KUKA KRL program: ho_st600_r1_bolha.src, ho_st600_r1_bolha.dat

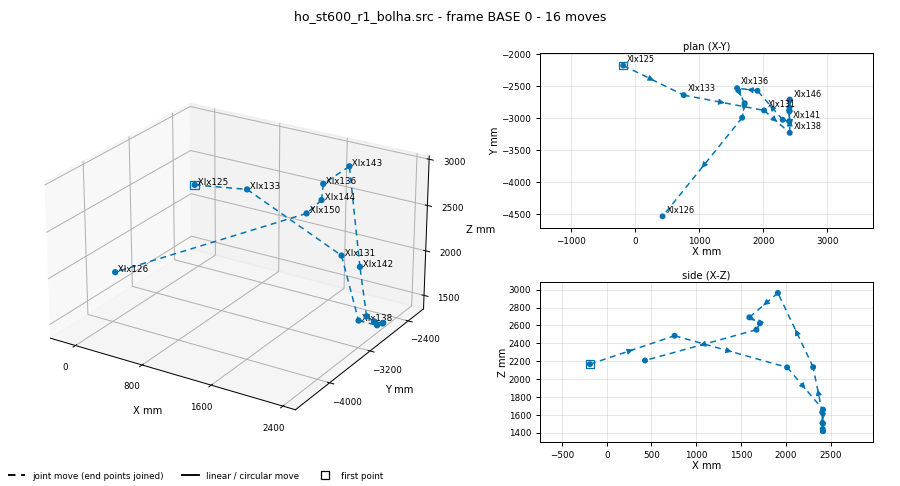
[picture p0: tool path of ho_st600_r1_bolha.src in frame BASE 0, 16 of 16 moves have a stored position in this frame; points joined in program order, loops and branches not executed]
--- ho_st600_r1_bolha.src ---
&ACCESS RVO1
&REL 2
&COMMENT Pega traseira ACCELO BOLHA
&PARAM DISKPATH = KRC:\R1\Program
DEF ho_st600_r1_Bolha( )
;FOLD INI
  ;FOLD BASISTECH INI
    GLOBAL INTERRUPT DECL 3 WHEN $STOPMESS==TRUE DO IR_STOPM ( )
    INTERRUPT ON 3
    BAS (#INITMOV,0 )
  ;ENDFOLD (BASISTECH INI)
;FOLD GRIPPERTECH INI
USER_GRP(0,DUMMY,DUMMY,GDEFAULT)
;ENDFOLD (GRIPPERTECH INI)
  ;FOLD USER INI
    ;Make your modifications here

  ;ENDFOLD (USER INI)
;ENDFOLD (INI)

; Caracterização dos meios de produção:
; Changes: Pega Traseira Accelo
; Versão Atual: 21/07/2015
; Name: P13.050-R1

chk_w7_wechs_ok ( )  ;CHECK GRIPPER TRASEIRO ACCELO


;FOLD PTP lx125 Vel=100 % PDAT8 Tool[7]:Painel Traseiro Accelo Base[0];%{PE}%R 8.2.20,%MKUKATPBASIS,%CMOVE,%VPTP,%P 1:PTP, 2:lx125, 3:, 5:100, 7:PDAT8
$BWDSTART=FALSE
PDAT_ACT=PPDAT8
FDAT_ACT=Flx125
BAS(#PTP_PARAMS,100)
PTP Xlx125
;ENDFOLD


;** SETUP DOS GRAMPOS PARA A BOLHA

;FOLD OUT 251 'Y2VR_FECHA_Accelo_Bolha' State=TRUE ;%{PE}%R 8.2.20,%MKUKATPBASIS,%COUT,%VOUTX,%P 2:251, 3:Y2VR_FECHA_Accelo_Bolha, 5:TRUE, 6:
$OUT[251]=TRUE
;ENDFOLD
;FOLD WAIT FOR ( IN 250 'Z2.1 - Grampo Avancado - Accelo Bolha' ) AND ( IN 252 'Z2.2 - Grampo Avancado - Accelo Bolha' );%{PE}%R 8.2.20,%MKUKATPBASIS,%CEXT_WAIT_FOR,%VEXT_WAIT_FOR,%P 2:, 4:, 5:$IN, 6:250, 7:Z2.1 - Grampo Avancado - Accelo Bolha, 9:AND, 10:, 12:, 13:$IN, 14:252, 15:Z2.2 - Grampo Avancado - Accelo Bolha, 17:
WAIT FOR  ( $IN[250] ) AND ( $IN[252] )
;ENDFOLD
;FOLD OUT 249 'Y1VR_FECHA_Accelo' State=TRUE ;%{PE}%R 8.2.20,%MKUKATPBASIS,%COUT,%VOUTX,%P 2:249, 3:Y1VR_FECHA_Accelo, 5:TRUE, 6:
$OUT[249]=TRUE
;ENDFOLD
;FOLD WAIT FOR ( IN 246 'Z1.2 - Grampo Avancado - Accelo - Traseiro' ) AND ( IN 248 'Z1.1 - Grampo Avancado - Accelo - Traseiro' );%{PE}%R 8.2.20,%MKUKATPBASIS,%CEXT_WAIT_FOR,%VEXT_WAIT_FOR,%P 2:, 4:, 5:$IN, 6:246, 7:Z1.2 - Grampo Avancado - Accelo - Traseiro, 9:AND, 10:, 12:, 13:$IN, 14:248, 15:Z1.1 - Grampo Avancado - Accelo - Traseiro, 17:
WAIT FOR  ( $IN[246] ) AND ( $IN[248] )
;ENDFOLD
;FOLD OUT 254 'Y3VR_RECUA_CILINDRO_Accelo/Bolha' State=TRUE ;%{PE}%R 8.2.20,%MKUKATPBASIS,%COUT,%VOUTX,%P 2:254, 3:Y3VR_RECUA_CILINDRO_Accelo/Bolha, 5:TRUE, 6:
$OUT[254]=TRUE
;ENDFOLD


;FOLD PTP lx133 Vel=100 % PDAT0 Tool[7]:Painel Traseiro Accelo Base[0];%{PE}%R 8.2.20,%MKUKATPBASIS,%CMOVE,%VPTP,%P 1:PTP, 2:lx133, 3:, 5:100, 7:PDAT0
$BWDSTART=FALSE
PDAT_ACT=PPDAT0
FDAT_ACT=Flx133
BAS(#PTP_PARAMS,100)
PTP Xlx133
;ENDFOLD

;FOLD WAIT FOR ( IN 253 'Z3.1 - Cilindro Recuado - Accelo' ) AND ( IN 255 'Z3.2 - Cilindro Recuado - Accelo' );%{PE}%R 8.2.20,%MKUKATPBASIS,%CEXT_WAIT_FOR,%VEXT_WAIT_FOR,%P 2:, 4:, 5:$IN, 6:253, 7:Z3.1 - Cilindro Recuado - Accelo, 9:AND, 10:, 12:, 13:$IN, 14:255, 15:Z3.2 - Cilindro Recuado - Accelo, 17:
WAIT FOR  ( $IN[253] ) AND ( $IN[255] )
;ENDFOLD
;FOLD OUT 251 'Y2VR_FECHA_Accelo_Bolha' State=FALSE ;%{PE}%R 8.2.20,%MKUKATPBASIS,%COUT,%VOUTX,%P 2:251, 3:Y2VR_FECHA_Accelo_Bolha, 5:FALSE, 6:
$OUT[251]=FALSE
;ENDFOLD
;FOLD WAIT Time=0.5 sec;%{PE}%R 8.2.20,%MKUKATPBASIS,%CWAIT,%VWAIT,%P 3:0.5
WAIT SEC 0.5
;ENDFOLD
;FOLD OUT 252 'Y2VR_ABRE_Accelo_Bolha' State=TRUE ;%{PE}%R 8.2.20,%MKUKATPBASIS,%COUT,%VOUTX,%P 2:252, 3:Y2VR_ABRE_Accelo_Bolha, 5:TRUE, 6:
$OUT[252]=TRUE
;ENDFOLD
;FOLD WAIT FOR ( IN 249 'Z2.1 - Grampo Recuado - Accelo Bolha' ) AND ( IN 251 'Z2.2 - Grampo Recuado - Accelo Bolha' );%{PE}%R 8.2.20,%MKUKATPBASIS,%CEXT_WAIT_FOR,%VEXT_WAIT_FOR,%P 2:, 4:, 5:$IN, 6:249, 7:Z2.1 - Grampo Recuado - Accelo Bolha, 9:AND, 10:, 12:, 13:$IN, 14:251, 15:Z2.2 - Grampo Recuado - Accelo Bolha, 17:
WAIT FOR  ( $IN[249] ) AND ( $IN[251] )
;ENDFOLD



;FOLD PTP lx131 CONT Vel=75 % PDAT14 Tool[7]:Painel Traseiro Accelo Base[0];%{PE}%R 8.2.20,%MKUKATPBASIS,%CMOVE,%VPTP,%P 1:PTP, 2:lx131, 3:C_DIS, 5:75, 7:PDAT14
$BWDSTART=FALSE
PDAT_ACT=PPDAT14
FDAT_ACT=Flx131
BAS(#PTP_PARAMS,75)
PTP Xlx131 C_DIS
;ENDFOLD

;FOLD PTP lx138 Vel=75 % PDAT21 Tool[7]:Painel Traseiro Accelo Base[0];%{PE}%R 8.2.20,%MKUKATPBASIS,%CMOVE,%VPTP,%P 1:PTP, 2:lx138, 3:, 5:75, 7:PDAT21
$BWDSTART=FALSE
PDAT_ACT=PPDAT21
FDAT_ACT=Flx138
BAS(#PTP_PARAMS,75)
PTP Xlx138
;ENDFOLD

;FOLD OUT 3352 'R1 busca traseira' State=TRUE ;%{PE}%R 8.2.20,%MKUKATPBASIS,%COUT,%VOUTX,%P 2:3352, 3:R1 busca traseira, 5:TRUE, 6:
$OUT[3352]=TRUE
;ENDFOLD
;FOLD WAIT FOR ( IN 3352 'Aguarda lib. Buscar traseira' );%{PE}%R 8.2.20,%MKUKATPBASIS,%CEXT_WAIT_FOR,%VEXT_WAIT_FOR,%P 2:, 4:, 5:$IN, 6:3352, 7:Aguarda lib. Buscar traseira, 9:
WAIT FOR  ( $IN[3352] )
;ENDFOLD
;FOLD OUT 3352 'R1 busca traseira' State=FALSE ;%{PE}%R 8.2.20,%MKUKATPBASIS,%COUT,%VOUTX,%P 2:3352, 3:R1 busca traseira, 5:FALSE, 6:
$OUT[3352]=FALSE
;ENDFOLD

;FOLD PTP lx124 CONT Vel=100 % PDAT7 Tool[7]:Painel Traseiro Accelo Base[0];%{PE}%R 8.2.20,%MKUKATPBASIS,%CMOVE,%VPTP,%P 1:PTP, 2:lx124, 3:C_DIS, 5:100, 7:PDAT7
$BWDSTART=FALSE
PDAT_ACT=PPDAT7
FDAT_ACT=Flx124
BAS(#PTP_PARAMS,100)
PTP Xlx124 C_DIS
;ENDFOLD
;FOLD PTP lx146 CONT Vel=100 % P_OLP5 Tool[7]:Painel Traseiro Accelo Base[0];%{PE}%R 8.2.20,%MKUKATPBASIS,%CMOVE,%VPTP,%P 1:PTP, 2:lx146, 3:C_DIS, 5:100, 7:P_OLP5
$BWDSTART=FALSE
PDAT_ACT=PP_OLP5
FDAT_ACT=Flx146
BAS(#PTP_PARAMS,100)
PTP Xlx146 C_DIS
;ENDFOLD

;FOLD OUT 3342 'Fora area externa' State=FALSE ;%{PE}%R 8.2.20,%MKUKATPBASIS,%COUT,%VOUTX,%P 2:3342, 3:Fora area externa, 5:FALSE, 6:
$OUT[3342]=FALSE
;ENDFOLD

;FOLD ; PONTO DE PEGA DA TRASEIRA ACCELO;%{PE}%R 8.2.20,%MKUKATPBASIS,%CCOMMENT,%VNORMAL,%P 2:PONTO  DE  PEGA  DA  TRASEIRA  ACCELO
;ENDFOLD
;FOLD LIN Xlx145  Vel=0.25 m/s L_OLP1 Tool[7]" " Base[0] ;%{PE}%R8.2,%MKUKATPBASIS,%CMOVE,%VLIN,%P 1:LIN, 2:lx145, 3:, 5:0.25, 7:L_OLP1
$BWDSTART = FALSE
LDAT_ACT= LL_OLP1
FDAT_ACT= Flx145
BAS(#CP_PARAMS,0.25)
LIN Xlx145
;ENDFOLD

IF (NOT(GHOST())) THEN
;FOLD WAIT FOR ( IN 241 'Presenca de peca 1 Accelo Bolha TRASEIRO' ) AND ( IN 242 'Presenca de peca 2 Accelo Bolha TRASEIRO' );%{PE}%R 8.2.20,%MKUKATPBASIS,%CEXT_WAIT_FOR,%VEXT_WAIT_FOR,%P 2:, 4:, 5:$IN, 6:241, 7:Presenca de peca 1 Accelo Bolha TRASEIRO, 9:AND, 10:, 12:, 13:$IN, 14:242, 15:Presenca de peca 2 Accelo Bolha TRASEIRO, 17:
WAIT FOR  ( $IN[241] ) AND ( $IN[242] )
;ENDFOLD
ENDIF


;FOLD OUT 252 'Y2VR_ABRE_Accelo_Bolha' State=FALSE ;%{PE}%R 8.2.20,%MKUKATPBASIS,%COUT,%VOUTX,%P 2:252, 3:Y2VR_ABRE_Accelo_Bolha, 5:FALSE, 6:
$OUT[252]=FALSE
;ENDFOLD

;FOLD OUT 251 'Y2VR_FECHA_Accelo_Bolha' State=TRUE ;%{PE}%R 8.2.20,%MKUKATPBASIS,%COUT,%VOUTX,%P 2:251, 3:Y2VR_FECHA_Accelo_Bolha, 5:TRUE, 6:
$OUT[251]=TRUE
;ENDFOLD
;FOLD WAIT FOR ( IN 250 'Z2.1 - Grampo Avancado - Accelo Bolha' ) AND ( IN 252 'Z2.2 - Grampo Avancado - Accelo Bolha' );%{PE}%R 8.2.20,%MKUKATPBASIS,%CEXT_WAIT_FOR,%VEXT_WAIT_FOR,%P 2:, 4:, 5:$IN, 6:250, 7:Z2.1 - Grampo Avancado - Accelo Bolha, 9:AND, 10:, 12:, 13:$IN, 14:252, 15:Z2.2 - Grampo Avancado - Accelo Bolha, 17:
WAIT FOR  ( $IN[250] ) AND ( $IN[252] )
;ENDFOLD

;FOLD OUT 248 'Liga_Sugador_Accelo_Bolha' State=TRUE ;%{PE}%R 8.2.20,%MKUKATPBASIS,%COUT,%VOUTX,%P 2:248, 3:Liga_Sugador_Accelo_Bolha, 5:TRUE, 6:
$OUT[248]=TRUE
;ENDFOLD
;FOLD WAIT FOR ( IN 259 'Vacuo1_Accelo_Bolha' ) AND ( IN 260 'Vacuo2_Accelo_Bolha' );%{PE}%R 8.2.20,%MKUKATPBASIS,%CEXT_WAIT_FOR,%VEXT_WAIT_FOR,%P 2:, 4:, 5:$IN, 6:259, 7:Vacuo1_Accelo_Bolha, 9:AND, 10:, 12:, 13:$IN, 14:260, 15:Vacuo2_Accelo_Bolha, 17:
WAIT FOR  ( $IN[259] ) AND ( $IN[260] )
;ENDFOLD

;FOLD OUT 257 'Liga_Magnetico_Accelo_Bolha' State=TRUE ;%{PE}%R 8.2.20,%MKUKATPBASIS,%COUT,%VOUTX,%P 2:257, 3:Liga_Magnetico_Accelo_Bolha, 5:TRUE, 6:
$OUT[257]=TRUE
;ENDFOLD




IF (NOT(GHOST())) THEN
ENDIF


;FOLD OUT 3349 'R1 pegou peça' State=TRUE ;%{PE}%R 8.2.20,%MKUKATPBASIS,%COUT,%VOUTX,%P 2:3349, 3:R1 pegou peça, 5:TRUE, 6:
$OUT[3349]=TRUE
;ENDFOLD
;FOLD OUT 3350 'Solicita lib sair magazine' State=TRUE ;%{PE}%R 8.2.20,%MKUKATPBASIS,%COUT,%VOUTX,%P 2:3350, 3:Solicita lib sair magazine, 5:TRUE, 6:
$OUT[3350]=TRUE
;ENDFOLD
;FOLD WAIT FOR ( IN 3349 'Aguarda lib sair magazine' );%{PE}%R 8.2.20,%MKUKATPBASIS,%CEXT_WAIT_FOR,%VEXT_WAIT_FOR,%P 2:, 4:, 5:$IN, 6:3349, 7:Aguarda lib sair magazine, 9:
WAIT FOR  ( $IN[3349] )
;ENDFOLD
;FOLD OUT 3350 'Solicita lib sair magazine' State=FALSE ;%{PE}%R 8.2.20,%MKUKATPBASIS,%COUT,%VOUTX,%P 2:3350, 3:Solicita lib sair magazine, 5:FALSE, 6:
$OUT[3350]=FALSE
;ENDFOLD

;FOLD LIN Xlx149  Vel=0.25 m/s L_OLP2 Tool[7]" " Base[0] ;%{PE}%R8.2,%MKUKATPBASIS,%CMOVE,%VLIN,%P 1:LIN, 2:lx149, 3:, 5:0.25, 7:L_OLP2
$BWDSTART = FALSE
LDAT_ACT= LL_OLP2
FDAT_ACT= Flx149
BAS(#CP_PARAMS,0.25)
LIN Xlx149
;ENDFOLD

;FOLD PTP lx134 CONT Vel=100 % PDAT17 Tool[7]:Painel Traseiro Accelo Base[0];%{PE}%R 8.2.20,%MKUKATPBASIS,%CMOVE,%VPTP,%P 1:PTP, 2:lx134, 3:C_DIS, 5:100, 7:PDAT17
$BWDSTART=FALSE
PDAT_ACT=PPDAT17
FDAT_ACT=Flx134
BAS(#PTP_PARAMS,100)
PTP Xlx134 C_DIS
;ENDFOLD


;FOLD PTP lx141 CONT Vel=100 % PDAT24 Tool[7]:Painel Traseiro Accelo Base[0];%{PE}%R 8.2.20,%MKUKATPBASIS,%CMOVE,%VPTP,%P 1:PTP, 2:lx141, 3:C_DIS, 5:100, 7:PDAT24
$BWDSTART=FALSE
PDAT_ACT=PPDAT24
FDAT_ACT=Flx141
BAS(#PTP_PARAMS,100)
PTP Xlx141 C_DIS
;ENDFOLD

;FOLD PTP lx142 CONT Vel=100 % PDAT25 Tool[7]:Painel Traseiro Accelo Base[0];%{PE}%R 8.2.20,%MKUKATPBASIS,%CMOVE,%VPTP,%P 1:PTP, 2:lx142, 3:C_DIS, 5:100, 7:PDAT25
$BWDSTART=FALSE
PDAT_ACT=PPDAT25
FDAT_ACT=Flx142
BAS(#PTP_PARAMS,100)
PTP Xlx142 C_DIS
;ENDFOLD


;FOLD PTP lx143 CONT Vel=100 % PDAT26 Tool[7]:Painel Traseiro Accelo Base[0];%{PE}%R 8.2.20,%MKUKATPBASIS,%CMOVE,%VPTP,%P 1:PTP, 2:lx143, 3:C_DIS, 5:100, 7:PDAT26
$BWDSTART=FALSE
PDAT_ACT=PPDAT26
FDAT_ACT=Flx143
BAS(#PTP_PARAMS,100)
PTP Xlx143 C_DIS
;ENDFOLD

;FOLD PTP lx136 CONT Vel=100 % PDAT19 Tool[7]:Painel Traseiro Accelo Base[0];%{PE}%R 8.2.20,%MKUKATPBASIS,%CMOVE,%VPTP,%P 1:PTP, 2:lx136, 3:C_DIS, 5:100, 7:PDAT19
$BWDSTART=FALSE
PDAT_ACT=PPDAT19
FDAT_ACT=Flx136
BAS(#PTP_PARAMS,100)
PTP Xlx136 C_DIS
;ENDFOLD

;FOLD PTP lx144 CONT Vel=100 % PDAT27 Tool[7]:Painel Traseiro Accelo Base[0];%{PE}%R 8.2.20,%MKUKATPBASIS,%CMOVE,%VPTP,%P 1:PTP, 2:lx144, 3:C_DIS, 5:100, 7:PDAT27
$BWDSTART=FALSE
PDAT_ACT=PPDAT27
FDAT_ACT=Flx144
BAS(#PTP_PARAMS,100)
PTP Xlx144 C_DIS
;ENDFOLD

;FOLD PTP lx150 CONT Vel=100 % P_OLP6 Tool[7]:Painel Traseiro Accelo Base[0];%{PE}%R8.2,%MKUKATPBASIS,%CMOVE,%VPTP,%P 1:PTP, 2:lx150, 3:C_DIS, 5:100, 7:P_OLP6
$BWDSTART = FALSE
PDAT_ACT= PP_OLP6
FDAT_ACT= Flx150
BAS(#PTP_PARAMS,100)
PTP Xlx150 C_DIS
;ENDFOLD
;FOLD PTP lx126 CONT Vel=100 % PDAT9 Tool[7]:Painel Traseiro Accelo Base[0];%{PE}%R 8.2.20,%MKUKATPBASIS,%CMOVE,%VPTP,%P 1:PTP, 2:lx126, 3:C_DIS, 5:100, 7:PDAT9
$BWDSTART=FALSE
PDAT_ACT=PPDAT9
FDAT_ACT=Flx126
BAS(#PTP_PARAMS,100)
PTP Xlx126 C_DIS
;ENDFOLD

;FOLD OUT 3349 'R1 Pegou peca' State=TRUE ;%{PE}%R 8.2.20,%MKUKATPBASIS,%COUT,%VOUTX,%P 2:3349, 3:R1 Pegou peca, 5:TRUE, 6:
$OUT[3349]=TRUE
;ENDFOLD
;FOLD OUT 3342 'Fora area externa' State=TRUE ;%{PE}%R 8.2.20,%MKUKATPBASIS,%COUT,%VOUTX,%P 2:3342, 3:Fora area externa, 5:TRUE, 6:
$OUT[3342]=TRUE
;ENDFOLD

END

--- ho_st600_r1_bolha.dat ---
&ACCESS RVO1
&REL 2
&COMMENT Pega traseira ACCELO BOLHA
&PARAM DISKPATH = KRC:\R1\Program
DEFDAT  ho_st600_r1_Bolha
;FOLD EXTERNAL DECLARATIONS;%{PE}%MKUKATPBASIS,%CEXT,%VCOMMON,%P
;FOLD GRIPPERTECH EXT
EXT  H50 (INT  :IN,INT  :IN,INT  :IN,GRP_TYP  :IN )
;ENDFOLD (GRIPPERTECH EXT)
;FOLD SPOTTECH EXT
EXT  USERSPOT (S_COMMAND  :IN,SPOT_TYPE  :IN )
;ENDFOLD (SPOTTECH EXT)
;FOLD BASISTECH EXT;%{PE}%MKUKATPBASIS,%CEXT,%VEXT,%P
EXT  BAS (BAS_COMMAND  :IN,REAL  :IN )
DECL INT SUCCESS
;ENDFOLD (BASISTECH EXT)
;FOLD USER EXT;%{E}%MKUKATPUSER,%CEXT,%VEXT,%P
;Make your modifications here

;ENDFOLD (USER EXT)
;ENDFOLD (EXTERNAL DECLARATIONS)

;# ============ START PATH : bh_p13050r1_ltc_02 =============
DECL FDAT Flx146={TOOL_NO 7,BASE_NO 0,IPO_FRAME #BASE,POINT2[] " ",TQ_STATE FALSE}
DECL PDAT PP_OLP5={VEL 100.0,ACC 100.0,APO_DIST 0.0,APO_MODE #CDIS}
DECL E6POS Xlx146={X 2414.24609,Y -2720.17798,Z 1419.953,A 89.8186417,B -64.6082993,C 179.921097,S 2,T 11,E1 -3712.55103,E2 0.0,E3 0.0,E4 0.0,E5 0.0,E6 0.0}
DECL FDAT Flx145={TOOL_NO 7,BASE_NO 0,IPO_FRAME #BASE,POINT2[] " ",TQ_STATE FALSE}
DECL E6POS Xlx145={X 2414.01489,Y -2707.33691,Z 1420.96399,A 89.5057068,B -64.9538422,C -179.770599,S 2,T 11,E1 -3712.55493,E2 0.0,E3 0.0,E4 0.0,E5 0.0,E6 0.0}
DECL LDAT LL_OLP1={VEL 0.25,ACC 100.0,APO_DIST 0.0,APO_FAC 0.0}
DECL FDAT Flx149={TOOL_NO 7,BASE_NO 0,IPO_FRAME #BASE,POINT2[] " "}
DECL E6POS Xlx149={X 2413.25488,Y -2887.86401,Z 1505.32397,A 89.5048828,B -64.9540634,C -179.769699,S 2,T 11,E1 -3712.55688,E2 0.0,E3 0.0,E4 0.0,E5 0.0,E6 0.0}
DECL LDAT LL_OLP2={VEL 0.25,ACC 100.0,APO_DIST 0.0,APO_FAC 0.0}
DECL FDAT Flx150={TOOL_NO 7,BASE_NO 0,IPO_FRAME #BASE,POINT2[] " "}
DECL PDAT PP_OLP6={VEL 100.0,ACC 100.0,APO_DIST 100.0,APO_MODE #CDIS}
DECL E6POS Xlx150={X 1671.224,Y -2991.78491,Z 2552.60889,A 44.4150009,B -75.0324783,C 129.688202,S 2,T 3,E1 -2192.70093,E2 0.0,E3 0.0,E4 0.0,E5 0.0,E6 0.0}
DECL BASIS_SUGG_T LAST_BASIS={POINT1[] "P0                      ",POINT2[] "P0                      ",CP_PARAMS[] "CPDAT0                  ",PTP_PARAMS[] "PDAT0                   ",CONT[] "                        ",CP_VEL[] "2.0                     ",PTP_VEL[] " 100                    ",SYNC_PARAMS[] "SYNCDAT                 ",SPL_NAME[] "S0                      "}
DECL GRP_SUGG_T LAST_GRP={NUMBER[] "5                       ",STATE[] "1                       ",PARAMS[] "GDAT3                   "}
DECL GRP_TYP GGDAT1={G_APO #NO,GRP_TIME 0.200000003,CTRL #OFF,DLY 0,DST 1}
DECL GRP_TYP GGDAT2={G_APO #NO,GRP_TIME 0.200000003,CTRL #OFF,DLY 0,DST 1}
DECL GRP_TYP GGDAT3={G_APO #NO,GRP_TIME 0.200000003,CTRL #OFF,DLY 0,DST 1}
DECL PDAT PPDAT7={VEL 100.0,ACC 100.0,APO_DIST 100.0,APO_MODE #CDIS}
DECL E6POS Xlx124={X 2410.65894,Y -2831.65405,Z 1444.37695,A 89.8383408,B -65.6056671,C -179.489899,S 2,T 11,E1 -3712.54712,E2 0.0,E3 0.0,E4 0.0,E5 0.0,E6 0.0}
DECL FDAT Flx124={TOOL_NO 7,BASE_NO 0,IPO_FRAME #BASE,POINT2[] " ",TQ_STATE FALSE}
DECL GRP_TYP GCONT={G_APO #YES,GRP_TIME 0.0,CTRL #OFF,DLY 0,DST 0}
DECL PDAT PPDAT8={VEL 100.0,ACC 100.0,APO_DIST 100.0,APO_MODE #CDIS}
DECL E6POS Xlx125={X -187.007996,Y -2175.83301,Z 2167.93994,A 48.8575897,B -57.0335617,C -142.841705,S 2,T 3,E1 -3715.35498,E2 0.0,E3 0.0,E4 0.0,E5 0.0,E6 0.0}
DECL FDAT Flx125={TOOL_NO 7,BASE_NO 0,IPO_FRAME #BASE,POINT2[] " ",TQ_STATE FALSE}
DECL E6POS XLX126={X 427.047913,Y -4533.16797,Z 2209.23389,A -73.5128708,B -78.8541565,C -161.542206,S 6,T 18,E1 -2536.18188,E2 0.0,E3 0.0,E4 0.0,E5 0.0,E6 0.0}
DECL FDAT Flx126={TOOL_NO 7,BASE_NO 0,IPO_FRAME #BASE,POINT2[] " ",TQ_STATE FALSE}
DECL PDAT PPDAT9={VEL 100.0,ACC 100.0,APO_DIST 100.0,APO_MODE #CDIS}
DECL GRP_TYP GGDAT4={G_APO #NO,GRP_TIME 0.200000003,CTRL #OFF,DLY 0,DST 1}
DECL PDAT PPDAT14={VEL 100.0,ACC 100.0,APO_DIST 100.0,APO_MODE #CDIS}
DECL E6POS Xlx131={X 2013.56104,Y -2877.54102,Z 2132.77197,A 86.6203995,B -62.3385391,C -177.631393,S 2,T 11,E1 -3712.88208,E2 0.0,E3 0.0,E4 0.0,E5 0.0,E6 0.0}
DECL FDAT Flx131={TOOL_NO 7,BASE_NO 0,IPO_FRAME #BASE,POINT2[] " ",TQ_STATE FALSE}
DECL PDAT PPDAT15={VEL 100.0,ACC 100.0,APO_DIST 100.0,APO_MODE #CDIS}
DECL E6POS Xlx132={X 757.784119,Y -2638.58398,Z 2485.66089,A 86.4221573,B -61.0999107,C -174.462006,S 2,T 11,E1 -3713.53003,E2 0.0,E3 0.0,E4 0.0,E5 0.0,E6 0.0}
DECL FDAT Flx132={TOOL_NO 7,BASE_NO 0,IPO_FRAME #BASE,POINT2[] " ",TQ_STATE FALSE}
DECL E6POS XLX134={X 2408.49707,Y -2891.43506,Z 1510.60596,A 89.8388672,B -65.7432404,C -179.910995,S 2,T 11,E1 -3712.552,E2 0.0,E3 0.0,E4 0.0,E5 0.0,E6 0.0}
DECL FDAT Flx134={TOOL_NO 7,BASE_NO 0,IPO_FRAME #BASE,POINT2[] " ",TQ_STATE FALSE}
DECL PDAT PPDAT17={VEL 100.0,ACC 100.0,APO_DIST 100.0,APO_MODE #CDIS}
DECL E6POS XLX135={X 2079.61499,Y -2528.86206,Z 2745.854,A 122.505203,B -59.1623993,C 117.408401,S 2,T 11,E1 -3182.0481,E2 0.0,E3 0.0,E4 0.0,E5 0.0,E6 0.0}
DECL FDAT Flx135={TOOL_NO 7,BASE_NO 0,IPO_FRAME #BASE,POINT2[] " ",TQ_STATE FALSE}
DECL PDAT PPDAT18={VEL 100.0,ACC 80.0,APO_DIST 80.0,APO_MODE #CDIS}
DECL E6POS XLX136={X 1592.48901,Y -2529.09399,Z 2691.021,A 97.9955597,B -64.183548,C 126.372902,S 2,T 11,E1 -2840.72803,E2 0.0,E3 0.0,E4 0.0,E5 0.0,E6 0.0}
DECL FDAT Flx136={TOOL_NO 7,BASE_NO 0,IPO_FRAME #BASE,POINT2[] " ",TQ_STATE FALSE}
DECL PDAT PPDAT19={VEL 100.0,ACC 80.0,APO_DIST 80.0,APO_MODE #CDIS}
DECL GRP_TYP GGDAT5={G_APO #NO,GRP_TIME 0.200000003,CTRL #OFF,DLY 0,DST 1}
DECL GRP_TYP GGDAT6={G_APO #NO,GRP_TIME 0.200000003,CTRL #OFF,DLY 0,DST 1}
DECL E6POS XLX138={X 2415.00293,Y -3227.64795,Z 1660.75,A 90.586319,B -65.2316589,C 179.779297,S 2,T 11,E1 -3712.55103,E2 0.0,E3 0.0,E4 0.0,E5 0.0,E6 0.0}
DECL FDAT Flx138={TOOL_NO 7,BASE_NO 0,IPO_FRAME #BASE,POINT2[] " ",TQ_STATE FALSE}
DECL PDAT PPDAT21={VEL 100.0,ACC 100.0,APO_DIST 100.0,APO_MODE #CDIS}
DECL E6POS XLX139={X 4758.36914,Y -8491.97852,Z -555.414185,A -47.7297401,B -59.6328011,C 156.117004,S 2,T 3,E1 -1239.23804,E2 0.0,E3 0.0,E4 0.0,E5 0.0,E6 0.0}
DECL FDAT Flx139={TOOL_NO 7,BASE_NO 2,IPO_FRAME #BASE,POINT2[] " ",TQ_STATE FALSE}
DECL PDAT PPDAT22={VEL 100.0,ACC 100.0,APO_DIST 100.0,APO_MODE #CDIS}
DECL E6POS XLX140={X 204.253403,Y 856.083374,Z 1303.87598,A 91.5418625,B -66.129509,C 142.588196,S 2,T 3,E1 -1796.73206,E2 0.0,E3 0.0,E4 0.0,E5 0.0,E6 0.0}
DECL FDAT Flx140={TOOL_NO 7,BASE_NO 0,IPO_FRAME #BASE,POINT2[] " ",TQ_STATE FALSE}
DECL PDAT PPDAT23={VEL 100.0,ACC 100.0,APO_DIST 100.0,APO_MODE #CDIS}
DECL E6POS XLX141={X 2405.90796,Y -3046.80591,Z 1630.87402,A 90.9038467,B -65.4751663,C 178.1483,S 2,T 11,E1 -3694.40308,E2 0.0,E3 0.0,E4 0.0,E5 0.0,E6 0.0}
DECL FDAT Flx141={TOOL_NO 7,BASE_NO 0,IPO_FRAME #BASE,POINT2[] " ",TQ_STATE FALSE}
DECL PDAT PPDAT24={VEL 100.0,ACC 100.0,APO_DIST 100.0,APO_MODE #CDIS}
DECL E6POS XLX142={X 2304.23999,Y -3023.67505,Z 2135.38403,A 119.099998,B -61.840229,C 145.630402,S 2,T 11,E1 -3668.80688,E2 0.0,E3 0.0,E4 0.0,E5 0.0,E6 0.0}
DECL FDAT Flx142={TOOL_NO 7,BASE_NO 0,IPO_FRAME #BASE,POINT2[] " ",TQ_STATE FALSE}
DECL PDAT PPDAT25={VEL 100.0,ACC 100.0,APO_DIST 100.0,APO_MODE #CDIS}
DECL E6POS XLX143={X 1911.12598,Y -2570.31494,Z 2963.18091,A 133.906494,B -53.9918289,C 105.7043,S 2,T 11,E1 -3211.09399,E2 0.0,E3 0.0,E4 0.0,E5 0.0,E6 0.0}
DECL FDAT Flx143={TOOL_NO 7,BASE_NO 0,IPO_FRAME #BASE,POINT2[] " ",TQ_STATE FALSE}
DECL PDAT PPDAT26={VEL 100.0,ACC 100.0,APO_DIST 100.0,APO_MODE #CDIS}
DECL E6POS XLX144={X 1710.67896,Y -2765.85498,Z 2624.51611,A 67.7690811,B -69.1723709,C 132.459198,S 2,T 11,E1 -2579.86108,E2 0.0,E3 0.0,E4 0.0,E5 0.0,E6 0.0}
DECL FDAT Flx144={TOOL_NO 7,BASE_NO 0,IPO_FRAME #BASE,POINT2[] " ",TQ_STATE FALSE}
DECL PDAT PPDAT27={VEL 100.0,ACC 80.0,APO_DIST 80.0,APO_MODE #CDIS}
DECL PDAT PPDAT0={VEL 100.0,ACC 100.0,APO_DIST 100.0,APO_MODE #CDIS}
DECL E6POS Xlx133={X 757.784119,Y -2638.58398,Z 2485.66089,A 86.4221573,B -61.0999107,C -174.462006,S 2,T 11,E1 -3713.53003,E2 0.0,E3 0.0,E4 0.0,E5 0.0,E6 0.0}
DECL FDAT Flx133={TOOL_NO 7,BASE_NO 0,IPO_FRAME #BASE,POINT2[] " ",TQ_STATE FALSE}
ENDDAT
